F_AssembleByteStream(
	pSrc:= ADR(SIR.Code), 
	SrcLen:= INT_TO_UDINT(LEN(SIR.Code)), 
	pDest:= ADR(SendTelegram), 
	DestLen:= SIZEOF(SendTelegram), 
	WritePointer:= WritePointer);

F_AssembleByteStream(
	pSrc:= ADR(SIR.TU_ID), 
	SrcLen:= INT_TO_UDINT(LEN(SIR.TU_ID)), 
	pDest:= ADR(SendTelegram), 
	DestLen:= SIZEOF(SendTelegram), 
	WritePointer:= WritePointer);	
	
F_AssembleByteStream(
	pSrc:= ADR(SIR.Counter1), 
	SrcLen:= INT_TO_UDINT(LEN(SIR.Counter1)), 
	pDest:= ADR(SendTelegram), 
	DestLen:= SIZEOF(SendTelegram), 
	WritePointer:= WritePointer);	
	
F_AssembleByteStream(
	pSrc:= ADR(SIR.Counter2), 
	SrcLen:= INT_TO_UDINT(LEN(SIR.Counter2)), 
	pDest:= ADR(SendTelegram), 
	DestLen:= SIZEOF(SendTelegram), 
	WritePointer:= WritePointer);	
	
F_AssembleByteStream(
	pSrc:= ADR(SIR.Counter3), 
	SrcLen:= INT_TO_UDINT(LEN(SIR.Counter3)), 
	pDest:= ADR(SendTelegram), 
	DestLen:= SIZEOF(SendTelegram), 
	WritePointer:= WritePointer);	
	
F_AssembleByteStream(
	pSrc:= ADR(SIR.Counter4), 
	SrcLen:= INT_TO_UDINT(LEN(SIR.Counter4)), 
	pDest:= ADR(SendTelegram), 
	DestLen:= SIZEOF(SendTelegram), 
	WritePointer:= WritePointer);	
	
F_AssembleByteStream(
	pSrc:= ADR(SIR.Counter5), 
	SrcLen:= INT_TO_UDINT(LEN(SIR.Counter5)), 
	pDest:= ADR(SendTelegram), 
	DestLen:= SIZEOF(SendTelegram), 
	WritePointer:= WritePointer);	

F_AssembleByteStream(
	pSrc:= ADR(SIR.ReturnCode), 
	SrcLen:= INT_TO_UDINT(LEN(SIR.ReturnCode)), 
	pDest:= ADR(SendTelegram), 
	DestLen:= SIZEOF(SendTelegram), 
	WritePointer:= WritePointer);


// Add to buffer of Base Driver
M_ProcessSIR := fbBaseDriver.M_SendAppData(
					mpSendData := ADR(SendTelegram),
					mSendDataLen := WritePointer);

// Forward to mirror channel
M_MirrorData(Data := ADR(SendTelegram), DataLen := WritePointer);
END_METHOD

METHOD PROTECTED M_ProcessSNR : BOOL
(**************************************************************************************
 * 	Application		:	BoxControl Framework
 *	Revision		:	$Revision: 404529 $
 *	Revision date	:	$Date: 2018-04-23 08:21:38 +0200 (Mo., 23 Apr 2018) $
 *	Last changed by	:	$Author: b7bolm $
 *	URL				:	$URL: http://almscdc.swisslog.com/repo/SWPD/Development/BoxControlFramework/20_Release/trunk/01_Software/BCF/BCF/JumpStart/20_Product/10_App/11_Com/10_Lib/10_Conv/12_MFCS/11_SIS/FB_SIS_MsgManager_6_1.TcPOU $
 *
 *	Purpose			:	Send SNR
 *
 * ------------------------------------------------------------------------------------
 *	Copyright Swisslog [IP AG], Switzerland. All rights reserved.
 * 
 * ------------------------------------------------------------------------------------
 *	
 * 	Revision History: 
 *
 * 	VERSION			DATE			INITIALS			DESCRIPTION
 *	0.1				01.01.2001		swl					Example
 *
 **************************************************************************************)
VAR_INPUT
 	meChannelSrc		: E_MFCS_Channel; // Source communicaton channel
	mpSNR				: POINTER TO ST_ITC_SNR; // Pointer to SNR
END_VAR
(**************************************************************************************************************
 	Check if a telegram needs to be send
***************************************************************************************************************)
// If settings allow sending a SNR 	
IF  Settings.Telegrams.SendSNR THEN
	// If the source of the request is this channel or is undefined
	IF meChannelSrc = Settings.MFCS_Channel OR
		meChannelSrc = E_MFCS_Channel.BEGIN_CHANNEL THEN
		;//Proceed
	ELSE // Source is a different MFCS Connection
		// Dont send a telegram		
		RETURN;
	END_IF	
ELSE
	// Dont send a telegram		
	RETURN;
END_IF

(**************************************************************************************************************
 	ITC - Map generic data to type
***************************************************************************************************************)
MEMCPY(destAddr := ADR(SNR_ITC), srcAddr := mpSNR, n := SIZEOF(SNR_ITC));

(**************************************************************************************************************
 	Formatting data
***************************************************************************************************************)

// Get SIS-Number 
SNR.Position := F_StuffString(
					InputString 	:= SNR_ITC.Position, 
					StringLength	:= SIS_6_1.POSITION_STRINGLENGTH, 
					StuffCharacter 	:= '0',
					LeftAligned		:= FALSE);

// Get TU-ID 
SNR.TU_ID := F_StuffString(
				InputString 	:= SNR_ITC.TU_ID, 
				StringLength	:= SIS_6_1.TU_ID_STRINGLENGTH, 
				StuffCharacter 	:= ' ',
				LeftAligned		:= FALSE);


// Get Error Code 
SNR.InfoCode := F_StuffString(
					InputString 	:= INT_TO_STRING(SNR_ITC.InfoCode), 
					StringLength	:= SIS_6_1.ERRORCODE_STRINGLENGTH, 
					StuffCharacter 	:= '0',
					LeftAligned		:= FALSE);
					
					
(**************************************************************************************************************
 	Build string and add to Base Driver
***************************************************************************************************************)
MEMSET(destAddr := ADR(SendTelegram), 0, SIZEOF(SendTelegram));
WritePointer := 0;

F_AssembleByteStream(
	pSrc:= ADR('SNR'), 
	SrcLen:= 3, 
	pDest:= ADR(SendTelegram), 
	DestLen:= SIZEOF(SendTelegram), 
	WritePointer:= WritePointer);
	
F_AssembleByteStream(
	pSrc:= ADR(SNR.Position), 
	SrcLen:= INT_TO_UDINT(LEN(SNR.Position)), 
	pDest:= ADR(SendTelegram), 
	DestLen:= SIZEOF(SendTelegram), 
	WritePointer:= WritePointer);

F_AssembleByteStream(
	pSrc:= ADR(SNR.TU_ID), 
	SrcLen:= INT_TO_UDINT(LEN(SNR.TU_ID)), 
	pDest:= ADR(SendTelegram), 
	DestLen:= SIZEOF(SendTelegram), 
	WritePointer:= WritePointer);
	
F_AssembleByteStream(
	pSrc:= ADR(SNR.InfoCode), 
	SrcLen:= INT_TO_UDINT(LEN(SNR.InfoCode)), 
	pDest:= ADR(SendTelegram), 
	DestLen:= SIZEOF(SendTelegram), 
	WritePointer:= WritePointer);

// Add to buffer of Base Driver
M_ProcessSNR := fbBaseDriver.M_SendAppData(
					mpSendData := ADR(SendTelegram),
					mSendDataLen := WritePointer);

// Forward to mirror channel
M_MirrorData(Data := ADR(SendTelegram), DataLen := WritePointer);
END_METHOD

METHOD PROTECTED M_ProcessSSR : BOOL
(**************************************************************************************
 * 	Application		:	BoxControl Framework
 *	Revision		:	$Revision: 404529 $
 *	Revision date	:	$Date: 2018-04-23 08:21:38 +0200 (Mo., 23 Apr 2018) $
 *	Last changed by	:	$Author: b7bolm $
 *	URL				:	$URL: http://almscdc.swisslog.com/repo/SWPD/Development/BoxControlFramework/20_Release/trunk/01_Software/BCF/BCF/JumpStart/20_Product/10_App/11_Com/10_Lib/10_Conv/12_MFCS/11_SIS/FB_SIS_MsgManager_6_1.TcPOU $
 *
 *	Purpose			:	Send SSR
 *
 * ------------------------------------------------------------------------------------
 *	Copyright Swisslog [IP AG], Switzerland. All rights reserved.
 * 
 * ------------------------------------------------------------------------------------
 *	
 * 	Revision History: 
 *
 * 	VERSION			DATE			INITIALS			DESCRIPTION
 *	0.1				01.01.2001		swl					Example
 *
 **************************************************************************************)
VAR_INPUT
 	meChannelSrc		: E_MFCS_Channel; // Source communicaton channel
	mpSSR				: POINTER TO ST_ITC_SSR; // Pointer to SSR
END_VAR
(**************************************************************************************************************
 	Check if a telegram needs to be send
***************************************************************************************************************)
// If settings allow sending a SSR 	
IF  Settings.Telegrams.SendSSR THEN
	// If the source of the request is this channel or is undefined
	IF meChannelSrc = Settings.MFCS_Channel OR
		meChannelSrc = E_MFCS_Channel.BEGIN_CHANNEL THEN
		;//Proceed
	ELSE // Source is a different MFCS Connection
		// Dont send a telegram		
		RETURN;
	END_IF	
ELSE
	// Dont send a telegram		
	RETURN;
END_IF

(**************************************************************************************************************
 	ITC - Map generic data to type
***************************************************************************************************************)
MEMCPY(destAddr := ADR(SSR_ITC), srcAddr := mpSSR, n := SIZEOF(SSR_ITC));

(**************************************************************************************************************
 	Formatting data
***************************************************************************************************************)
// Get Subsystem name 
SSR.SubsystemName := F_StuffString(
						InputString 	:= SSR_ITC.SubsystemName, 
						StringLength	:= SIS_6_1.POSITION_STRINGLENGTH, 
						StuffCharacter 	:= '0',
						LeftAligned		:= FALSE);

// Get Mode 
SSR.Mode := INT_TO_STRING(SSR_ITC.eMode);

// Get system info
SSR.State := INT_TO_STRING(SSR_ITC.eState);

// Get system info
SSR.SystemInfo := INT_TO_STRING(SSR_ITC.eSystemInfo);

// Get ErrorState 
SSR.ErrorState := INT_TO_STRING(SSR_ITC.eErrorState);

// Get ErrorCode 
SSR.ErrorCode := F_StuffString(
					InputString 	:= INT_TO_STRING(SSR_ITC.eErrorCode), 
					StringLength	:= SIS_6_1.ERRORCODE_STRINGLENGTH, 
					StuffCharacter 	:= '0',
					LeftAligned		:= FALSE);

// Get ErrorType 
SSR.ErrorType := INT_TO_STRING(SSR_ITC.eErrorType);

// Get ErrorInformation 
SSR.ErrorInformation := F_StuffString(
							InputString 	:= SSR_ITC.ErrorInformation, 
							StringLength	:= SIS_6_1.ERRORINFORMATION_STRINGLENGTH, 
							StuffCharacter 	:= ' ',
							LeftAligned		:= TRUE);

// Get Variable 
SSR.Variable := F_StuffString(
					InputString 	:= DINT_TO_STRING(SSR_ITC.Variable), 
					StringLength	:= SIS_6_1.CONTROLVARIABLE_STRINGLENGTH, 
					StuffCharacter 	:= '0',
					LeftAligned		:= FALSE);

// Get Error Code 
SSR.ReturnCode := F_StuffString(
					InputString 	:= INT_TO_STRING(SSR_ITC.eReturnCode), 
					StringLength	:= SIS_6_1.ERRORCODE_STRINGLENGTH, 
					StuffCharacter 	:= '0',
					LeftAligned		:= FALSE);


(**************************************************************************************************************
 	Build string and add to Base Driver
***************************************************************************************************************)
MEMSET(destAddr := ADR(SendTelegram), 0, SIZEOF(SendTelegram));
WritePointer := 0;

F_AssembleByteStream(
	pSrc:= ADR('SSR'), 
	SrcLen:= 3, 
	pDest:= ADR(SendTelegram), 
	DestLen:= SIZEOF(SendTelegram), 
	WritePointer:= WritePointer);
	
F_AssembleByteStream(
	pSrc:= ADR(SSR.SubsystemName), 
	SrcLen:= INT_TO_UDINT(LEN(SSR.SubsystemName)), 
	pDest:= ADR(SendTelegram), 
	DestLen:= SIZEOF(SendTelegram), 
	WritePointer:= WritePointer);

F_AssembleByteStream(
	pSrc:= ADR(SSR.Mode), 
	SrcLen:= INT_TO_UDINT(LEN(SSR.Mode)), 
	pDest:= ADR(SendTelegram), 
	DestLen:= SIZEOF(SendTelegram), 
	WritePointer:= WritePointer);	

F_AssembleByteStream(
	pSrc:= ADR(SSR.State), 
	SrcLen:= INT_TO_UDINT(LEN(SSR.State)), 
	pDest:= ADR(SendTelegram), 
	DestLen:= SIZEOF(SendTelegram), 
	WritePointer:= WritePointer);	

F_AssembleByteStream(
	pSrc:= ADR(SSR.SystemInfo), 
	SrcLen:= INT_TO_UDINT(LEN(SSR.SystemInfo)), 
	pDest:= ADR(SendTelegram), 
	DestLen:= SIZEOF(SendTelegram), 
	WritePointer:= WritePointer);	
	
F_AssembleByteStream(
	pSrc:= ADR(SSR.ErrorState), 
	SrcLen:= INT_TO_UDINT(LEN(SSR.ErrorState)), 
	pDest:= ADR(SendTelegram), 
	DestLen:= SIZEOF(SendTelegram), 
	WritePointer:= WritePointer);

F_AssembleByteStream(
	pSrc:= ADR(SSR.ErrorCode), 
	SrcLen:= INT_TO_UDINT(LEN(SSR.ErrorCode)), 
	pDest:= ADR(SendTelegram), 
	DestLen:= SIZEOF(SendTelegram), 
	WritePointer:= WritePointer);

F_AssembleByteStream(
	pSrc:= ADR(SSR.ErrorType), 
	SrcLen:= INT_TO_UDINT(LEN(SSR.ErrorType)), 
	pDest:= ADR(SendTelegram), 
	DestLen:= SIZEOF(SendTelegram), 
	WritePointer:= WritePointer);
	
F_AssembleByteStream(
	pSrc:= ADR(SSR.ErrorInformation), 
	SrcLen:= INT_TO_UDINT(LEN(SSR.ErrorInformation)), 
	pDest:= ADR(SendTelegram), 
	DestLen:= SIZEOF(SendTelegram), 
	WritePointer:= WritePointer);
	
F_AssembleByteStream(
	pSrc:= ADR(SSR.Variable), 
	SrcLen:= INT_TO_UDINT(LEN(SSR.Variable)), 
	pDest:= ADR(SendTelegram), 
	DestLen:= SIZEOF(SendTelegram), 
	WritePointer:= WritePointer);
	
F_AssembleByteStream(
	pSrc:= ADR(SSR.ReturnCode), 
	SrcLen:= INT_TO_UDINT(LEN(SSR.ReturnCode)), 
	pDest:= ADR(SendTelegram), 
	DestLen:= SIZEOF(SendTelegram), 
	WritePointer:= WritePointer);

// Add to buffer of Base Driver
M_ProcessSSR := fbBaseDriver.M_SendAppData(
					mpSendData := ADR(SendTelegram),
					mSendDataLen := WritePointer);

// Forward to mirror channel
M_MirrorData(Data := ADR(SendTelegram), DataLen := WritePointer);
END_METHOD

METHOD PROTECTED M_ProcessTDR : BOOL
(**************************************************************************************
 * 	Application		:	BoxControl Framework
 *	Revision		:	$Revision: 404529 $
 *	Revision date	:	$Date: 2018-04-23 08:21:38 +0200 (Mo., 23 Apr 2018) $
 *	Last changed by	:	$Author: b7bolm $
 *	URL				:	$URL: http://almscdc.swisslog.com/repo/SWPD/Development/BoxControlFramework/20_Release/trunk/01_Software/BCF/BCF/JumpStart/20_Product/10_App/11_Com/10_Lib/10_Conv/12_MFCS/11_SIS/FB_SIS_MsgManager_6_1.TcPOU $
 *
 *	Purpose			:	Send TDR
 *
 * ------------------------------------------------------------------------------------
 *	Copyright Swisslog [IP AG], Switzerland. All rights reserved.
 * 
 * ------------------------------------------------------------------------------------
 *	
 * 	Revision History: 
 *
 * 	VERSION			DATE			INITIALS			DESCRIPTION
 *	0.1				01.01.2001		swl					Example
 *
 **************************************************************************************)
VAR_INPUT
 	meChannelSrc		: E_MFCS_Channel; // Source communicaton channel
	mpTDR				: POINTER TO ST_ITC_TDR; // Pointer to TDR
END_VAR
(**************************************************************************************************************
 	Check if a telegram needs to be send
***************************************************************************************************************)
// If settings allow sending a TDR 	
IF  Settings.Telegrams.SendTDR THEN
	// If the source of the request is this channel or is undefined
	IF meChannelSrc = Settings.MFCS_Channel OR
		meChannelSrc = E_MFCS_Channel.BEGIN_CHANNEL THEN
		;//Proceed
	ELSE // Source is a different MFCS Connection
		// Dont send a telegram		
		RETURN;
	END_IF	
ELSE
	// Dont send a telegram		
	RETURN;
END_IF

(**************************************************************************************************************
 	ITC - Map generic data to type
***************************************************************************************************************)
MEMCPY(destAddr := ADR(TDR_ITC), srcAddr := mpTDR, n := SIZEOF(TDR_ITC));

(**************************************************************************************************************
 	Formatting data
***************************************************************************************************************)
// Get SIS-Number 
TDR.Position := F_StuffString(
					InputString 	:= TDR_ITC.Position, 
					StringLength	:= SIS_6_1.POSITION_STRINGLENGTH, 
					StuffCharacter 	:= '0',
					LeftAligned		:= FALSE);

// Get TU-ID 
TDR.TU_ID := F_StuffString(
				InputString 	:= TDR_ITC.TU_ID, 
				StringLength	:= SIS_6_1.TU_ID_STRINGLENGTH, 
				StuffCharacter 	:= ' ',
				LeftAligned		:= FALSE);
					
// Get Assignment 
TDR.AssignmentID := F_StuffString(
						InputString 	:= UDINT_TO_STRING(TDR_ITC.AssignmentID), 
						StringLength	:= SIS_6_1.ASSIGNMENT_ID_STRINGLENGTH, 
						StuffCharacter 	:= '0',
						LeftAligned		:= FALSE);

// Get MSG Sequence 
TDR.MsgSequence := 	F_StuffString(
						InputString 	:= INT_TO_STRING(TDR_ITC.MsgSequence), 
						StringLength	:= SIS_6_1.MSG_SEQUENCE_STRINGLENGTH, 
						StuffCharacter 	:= '0',
						LeftAligned		:= FALSE);

// Get return Code 
TDR.ReturnCode := F_StuffString(
					InputString 	:= INT_TO_STRING(TDR_ITC.ReturnCode), 
					StringLength	:= SIS_6_1.ERRORCODE_STRINGLENGTH, 
					StuffCharacter 	:= '0',
					LeftAligned		:= FALSE);



(**************************************************************************************************************
 	Build string and add to Base Driver
***************************************************************************************************************)
MEMSET(destAddr := ADR(SendTelegram), 0, SIZEOF(SendTelegram));
WritePointer := 0;

F_AssembleByteStream(
	pSrc:= ADR('TDR'), 
	SrcLen:= 3, 
	pDest:= ADR(SendTelegram), 
	DestLen:= SIZEOF(SendTelegram), 
	WritePointer:= WritePointer);
	
F_AssembleByteStream(
	pSrc:= ADR(TDR.Position), 
	SrcLen:= INT_TO_UDINT(LEN(TDR.Position)), 
	pDest:= ADR(SendTelegram), 
	DestLen:= SIZEOF(SendTelegram), 
	WritePointer:= WritePointer);

F_AssembleByteStream(
	pSrc:= ADR(TDR.TU_ID), 
	SrcLen:= INT_TO_UDINT(LEN(TDR.TU_ID)), 
	pDest:= ADR(SendTelegram), 
	DestLen:= SIZEOF(SendTelegram), 
	WritePointer:= WritePointer);
	
F_AssembleByteStream(
	pSrc:= ADR(TDR.AssignmentID), 
	SrcLen:= INT_TO_UDINT(LEN(TDR.AssignmentID)), 
	pDest:= ADR(SendTelegram), 
	DestLen:= SIZEOF(SendTelegram), 
	WritePointer:= WritePointer);
	
F_AssembleByteStream(
	pSrc:= ADR(TDR.MsgSequence), 
	SrcLen:= INT_TO_UDINT(LEN(TDR.MsgSequence)), 
	pDest:= ADR(SendTelegram), 
	DestLen:= SIZEOF(SendTelegram), 
	WritePointer:= WritePointer);	
	
F_AssembleByteStream(
	pSrc:= ADR(TDR.ReturnCode), 
	SrcLen:= INT_TO_UDINT(LEN(TDR.ReturnCode)), 
	pDest:= ADR(SendTelegram), 
	DestLen:= SIZEOF(SendTelegram), 
	WritePointer:= WritePointer);	

// Add to buffer of Base Driver
M_ProcessTDR := fbBaseDriver.M_SendAppData(
					mpSendData := ADR(SendTelegram),
					mSendDataLen := WritePointer);

// Forward to mirror channel
M_MirrorData(Data := ADR(SendTelegram), DataLen := WritePointer);
END_METHOD

METHOD PROTECTED M_ProcessTTC : BOOL
(**************************************************************************************
 * 	Application		:	BoxControl Framework
 *	Revision		:	$Revision: 404529 $
 *	Revision date	:	$Date: 2018-04-23 08:21:38 +0200 (Mo., 23 Apr 2018) $
 *	Last changed by	:	$Author: b7bolm $
 *	URL				:	$URL: http://almscdc.swisslog.com/repo/SWPD/Development/BoxControlFramework/20_Release/trunk/01_Software/BCF/BCF/JumpStart/20_Product/10_App/11_Com/10_Lib/10_Conv/12_MFCS/11_SIS/FB_SIS_MsgManager_6_1.TcPOU $
 *
 *	Purpose			:	Send TTC
 *
 * ------------------------------------------------------------------------------------
 *	Copyright Swisslog [IP AG], Switzerland. All rights reserved.
 * 
 * ------------------------------------------------------------------------------------
 *	
 * 	Revision History: 
 *
 * 	VERSION			DATE			INITIALS			DESCRIPTION
 *	0.1				01.01.2001		swl					Example
 *
 **************************************************************************************)
VAR_INPUT
 	meChannelSrc		: E_MFCS_Channel; // Source communicaton channel
	mpTTC				: POINTER TO ST_ITC_TTC; // Pointer to TTC
END_VAR
(**************************************************************************************************************
 	Check if a telegram needs to be send
***************************************************************************************************************)
// If settings allow sending a TTC 	
IF  Settings.Telegrams.SendTTC THEN
	// If the source of the request is this channel or is undefined
	IF meChannelSrc = Settings.MFCS_Channel OR
		meChannelSrc = E_MFCS_Channel.BEGIN_CHANNEL THEN
		;//Proceed
	ELSE // Source is a different MFCS Connection
		// Dont send a telegram		
		RETURN;
	END_IF	
ELSE
	// Dont send a telegram		
	RETURN;
END_IF

(**************************************************************************************************************
 	ITC - Map generic data to type
***************************************************************************************************************)
MEMCPY(destAddr := ADR(TTC_ITC), srcAddr := mpTTC, n := SIZEOF(TTC_ITC));

(**************************************************************************************************************
 	Formatting data
***************************************************************************************************************)
// Get SIS-Number 
TTC.Position := F_StuffString(
					InputString 	:= TTC_ITC.Position, 
					StringLength	:= SIS_6_1.POSITION_STRINGLENGTH, 
					StuffCharacter 	:= '0',
					LeftAligned		:= FALSE);

// Get TU-DataIndex 
TTC.TU_DataIndex := F_StuffString(
						InputString 	:= DINT_TO_STRING(TTC_ITC.TU_DataIndex), 
						StringLength	:= SIS_6_1.TU_DATAINDEX_STRINGLENGTH, 
						StuffCharacter 	:= '0',
						LeftAligned		:= FALSE);

// Get MSG Sequence 
TTC.MsgSequence := F_StuffString(
						InputString 	:= INT_TO_STRING(TTC_ITC.MsgSequence), 
						StringLength	:= SIS_6_1.MSG_SEQUENCE_STRINGLENGTH, 
						StuffCharacter 	:= '0',
						LeftAligned		:= FALSE);

// Get TU-ID 
TTC.TU_ID := F_StuffString(
				InputString 	:= TTC_ITC.TU_ID, 
				StringLength	:= SIS_6_1.TU_ID_STRINGLENGTH, 
				StuffCharacter 	:= ' ',
				LeftAligned		:= FALSE);
				
// Get Assignment 
TTC.AssignmentID := F_StuffString(
						InputString 	:= UDINT_TO_STRING(TTC_ITC.AssignmentID), 
						StringLength	:= SIS_6_1.ASSIGNMENT_ID_STRINGLENGTH, 
						StuffCharacter 	:= '0',
						LeftAligned		:= FALSE);

// Get Error Code 
TTC.ReturnCode := F_StuffString(
					InputString 	:= INT_TO_STRING(TTC_ITC.ReturnCode), 
					StringLength	:= SIS_6_1.ERRORCODE_STRINGLENGTH, 
					StuffCharacter 	:= '0',
					LeftAligned		:= FALSE);

(**************************************************************************************************************
 	Build string and add to Base Driver
***************************************************************************************************************)
MEMSET(destAddr := ADR(SendTelegram), 0, SIZEOF(SendTelegram));
WritePointer := 0;

F_AssembleByteStream(
	pSrc:= ADR('TTC'), 
	SrcLen:= 3, 
	pDest:= ADR(SendTelegram), 
	DestLen:= SIZEOF(SendTelegram), 
	WritePointer:= WritePointer);
	
F_AssembleByteStream(
	pSrc:= ADR(TTC.Position), 
	SrcLen:= INT_TO_UDINT(LEN(TTC.Position)), 
	pDest:= ADR(SendTelegram), 
	DestLen:= SIZEOF(SendTelegram), 
	WritePointer:= WritePointer);
	
F_AssembleByteStream(
	pSrc:= ADR(TTC.TU_DataIndex), 
	SrcLen:= INT_TO_UDINT(LEN(TTC.TU_DataIndex)), 
	pDest:= ADR(SendTelegram), 
	DestLen:= SIZEOF(SendTelegram), 
	WritePointer:= WritePointer);
	
F_AssembleByteStream(
	pSrc:= ADR(TTC.MsgSequence), 
	SrcLen:= INT_TO_UDINT(LEN(TTC.MsgSequence)), 
	pDest:= ADR(SendTelegram), 
	DestLen:= SIZEOF(SendTelegram), 
	WritePointer:= WritePointer);

F_AssembleByteStream(
	pSrc:= ADR(TTC.TU_ID), 
	SrcLen:= INT_TO_UDINT(LEN(TTC.TU_ID)), 
	pDest:= ADR(SendTelegram), 
	DestLen:= SIZEOF(SendTelegram), 
	WritePointer:= WritePointer);

F_AssembleByteStream(
	pSrc:= ADR(TTC.AssignmentID), 
	SrcLen:= INT_TO_UDINT(LEN(TTC.AssignmentID)), 
	pDest:= ADR(SendTelegram), 
	DestLen:= SIZEOF(SendTelegram), 
	WritePointer:= WritePointer);

F_AssembleByteStream(
	pSrc:= ADR(TTC.ReturnCode), 
	SrcLen:= INT_TO_UDINT(LEN(TTC.ReturnCode)), 
	pDest:= ADR(SendTelegram), 
	DestLen:= SIZEOF(SendTelegram), 
	WritePointer:= WritePointer);

// Add to buffer of Base Driver
M_ProcessTTC := fbBaseDriver.M_SendAppData(
					mpSendData := ADR(SendTelegram),
					mSendDataLen := WritePointer);

// Forward to mirror channel
M_MirrorData(Data := ADR(SendTelegram), DataLen := WritePointer);
END_METHOD

METHOD PROTECTED M_ProcessTTQ : BOOL
(**************************************************************************************
 * 	Application		:	BoxControl Framework
 *	Revision		:	$Revision: 404529 $
 *	Revision date	:	$Date: 2018-04-23 08:21:38 +0200 (Mo., 23 Apr 2018) $
 *	Last changed by	:	$Author: b7bolm $
 *	URL				:	$URL: http://almscdc.swisslog.com/repo/SWPD/Development/BoxControlFramework/20_Release/trunk/01_Software/BCF/BCF/JumpStart/20_Product/10_App/11_Com/10_Lib/10_Conv/12_MFCS/11_SIS/FB_SIS_MsgManager_6_1.TcPOU $
 *
 *	Purpose			:	Send TTQ
 *
 * ------------------------------------------------------------------------------------
 *	Copyright Swisslog [IP AG], Switzerland. All rights reserved.
 * 
 * ------------------------------------------------------------------------------------
 *	
 * 	Revision History: 
 *
 * 	VERSION			DATE			INITIALS			DESCRIPTION
 *	0.1				01.01.2001		swl					Example
 *
 **************************************************************************************)
VAR_INPUT
 	meChannelSrc		: E_MFCS_Channel; // Source communicaton channel
	mpTTQ				: POINTER TO ST_ITC_TTQ; // Pointer to TTQ
END_VAR
(**************************************************************************************************************
 	Check if a telegram needs to be send
***************************************************************************************************************)
// If settings allow sending a TTQ 	
IF  Settings.Telegrams.SendTTQ THEN
	// If the source of the request is this channel or is undefined
	IF meChannelSrc = Settings.MFCS_Channel OR
		meChannelSrc = E_MFCS_Channel.BEGIN_CHANNEL THEN
		;//Proceed
	ELSE // Source is a different MFCS Connection
		// Dont send a telegram		
		RETURN;
	END_IF	
ELSE
	// Dont send a telegram		
	RETURN;
END_IF

(**************************************************************************************************************
 	ITC - Map generic data to type
***************************************************************************************************************)
MEMCPY(destAddr := ADR(TTQ_ITC), srcAddr := mpTTQ, n := SIZEOF(TTQ_ITC));

(**************************************************************************************************************
 	Formatting data
***************************************************************************************************************)
// Get SIS-Number 
TTQ.Position := F_StuffString(
					InputString 	:= TTQ_ITC.Position, 
					StringLength	:= SIS_6_1.POSITION_STRINGLENGTH, 
					StuffCharacter 	:= '0',
					LeftAligned		:= FALSE);

// Get TU-DataIndex 
TTQ.TU_DataIndex := F_StuffString(
						InputString 	:= DINT_TO_STRING(TTQ_ITC.TU_DataIndex), 
						StringLength	:= SIS_6_1.TU_DATAINDEX_STRINGLENGTH, 
						StuffCharacter 	:= '0',
						LeftAligned		:= FALSE);

// Get TU-ID 
TTQ.TU_ID := F_StuffString(
				InputString 	:= TTQ_ITC.TU_ID, 
				StringLength	:= SIS_6_1.TU_ID_STRINGLENGTH, 
				StuffCharacter 	:= ' ',
				LeftAligned		:= FALSE);

// Get Number of TT's 
TTQ.NbrOfTT :=  F_StuffString(
						InputString 	:= INT_TO_STRING(TTQ_ITC.NbrOfTT), 
						StringLength	:= SIS_6_1.TTQ_NUMBER_OF_TT_STRINGLENGTH, 
						StuffCharacter 	:= '0',
						LeftAligned		:= FALSE);

// Get Label Length						
TTQ.Label := F_StuffString(
				InputString 	:= TTQ_ITC.Label, 
				StringLength	:= Conveyor.LABEL_LENGTH, 
				StuffCharacter 	:= '-',
				LeftAligned		:= FALSE);

(**************************************************************************************************************
 	Build string and add to Base Driver
***************************************************************************************************************)
MEMSET(destAddr := ADR(SendTelegram), 0, SIZEOF(SendTelegram));
WritePointer := 0;

F_AssembleByteStream(
	pSrc:= ADR('TTQ'), 
	SrcLen:= 3, 
	pDest:= ADR(SendTelegram), 
	DestLen:= SIZEOF(SendTelegram), 
	WritePointer:= WritePointer);
	
F_AssembleByteStream(
	pSrc:= ADR(TTQ .Position), 
	SrcLen:= INT_TO_UDINT(LEN(TTQ.Position)), 
	pDest:= ADR(SendTelegram), 
	DestLen:= SIZEOF(SendTelegram), 
	WritePointer:= WritePointer);

F_AssembleByteStream(
	pSrc:= ADR(TTQ.TU_DataIndex), 
	SrcLen:= INT_TO_UDINT(LEN(TTQ.TU_DataIndex)), 
	pDest:= ADR(SendTelegram), 
	DestLen:= SIZEOF(SendTelegram), 
	WritePointer:= WritePointer);
	
F_AssembleByteStream(
	pSrc:= ADR(TTQ.TU_ID), 
	SrcLen:= INT_TO_UDINT(LEN(TTQ.TU_ID)), 
	pDest:= ADR(SendTelegram), 
	DestLen:= SIZEOF(SendTelegram), 
	WritePointer:= WritePointer);
	
F_AssembleByteStream(
	pSrc:= ADR(TTQ.NbrOfTT), 
	SrcLen:= INT_TO_UDINT(LEN(TTQ.NbrOfTT)), 
	pDest:= ADR(SendTelegram), 
	DestLen:= SIZEOF(SendTelegram), 
	WritePointer:= WritePointer);
	
F_AssembleByteStream(
	pSrc:= ADR(TTQ.Label), 
	SrcLen:= INT_TO_UDINT(LEN(TTQ.Label)), 
	pDest:= ADR(SendTelegram), 
	DestLen:= SIZEOF(SendTelegram), 
	WritePointer:= WritePointer);	


// Add to buffer of Base Driver
M_ProcessTTQ := fbBaseDriver.M_SendAppData(
					mpSendData := ADR(SendTelegram),
					mSendDataLen := WritePointer);

// Forward to mirror channel
M_MirrorData(Data := ADR(SendTelegram), DataLen := WritePointer);
END_METHOD

METHOD PROTECTED M_ProcessTUR : BOOL
(**************************************************************************************
 * 	Application		:	BoxControl Framework
 *	Revision		:	$Revision: 415970 $
 *	Revision date	:	$Date: 2018-10-24 16:08:06 +0200 (Mi., 24 Okt 2018) $
 *	Last changed by	:	$Author: d7herza $
 *	URL				:	$URL: http://almscdc.swisslog.com/repo/SWPD/Development/BoxControlFramework/20_Release/branches/R1.5.x/01_Software/BCF/BCF/JumpStart/20_Product/10_App/11_Com/10_Lib/10_Conv/12_MFCS/11_SIS/FB_SIS_MsgManager_6_1.TcPOU $
 *
 *	Purpose			:	Send TUR
 *
 * ------------------------------------------------------------------------------------
 *	Copyright Swisslog [IP AG], Switzerland. All rights reserved.
 * 
 * ------------------------------------------------------------------------------------
 *	
 * 	Revision History: 
 *
 * 	VERSION			DATE			INITIALS			DESCRIPTION
 *	0.1				01.01.2001		swl					Example
 *
 *************************************************************************************)
VAR_INPUT
 	meChannelSrc		: E_MFCS_Channel; // Source communicaton channel
	mpTUR				: POINTER TO ST_ITC_TUR; // Pointer to TUR
END_VAR

VAR
	DestinationIdx			: INT; // Iterator
END_VAR
(**************************************************************************************************************
 	Check if a telegram needs to be send
***************************************************************************************************************)
// If settings allow sending a TUR 	
IF  Settings.Telegrams.SendTUR THEN
	// If the source of the request is this channel or is undefined
	IF meChannelSrc = Settings.MFCS_Channel OR
		meChannelSrc = E_MFCS_Channel.BEGIN_CHANNEL THEN
		;//Proceed
	ELSE // Source is a different MFCS Connection
		// Dont send a telegram		
		RETURN;
	END_IF	
ELSE
	// Dont send a telegram		
	RETURN;
END_IF

(**************************************************************************************************************
 	ITC - Map generic data to type
***************************************************************************************************************)
MEMCPY(destAddr := ADR(TUR_ITC), srcAddr := mpTUR, n := SIZEOF(TUR_ITC));

(**************************************************************************************************************
 	Formatting data
***************************************************************************************************************)
// Get SIS-Number 
TUR.Position := F_StuffString(
					InputString 	:= TUR_ITC.Position, 
					StringLength	:= SIS_6_1.POSITION_STRINGLENGTH, 
					StuffCharacter 	:= '0',
					LeftAligned		:= FALSE);
				
// Get TU-Data index
TUR.TU_DataIndex := F_StuffString(
				InputString 	:= DINT_TO_STRING(TUR_ITC.TU_DataIndex), 
				StringLength	:= SIS_6_1.TU_DATAINDEX_STRINGLENGTH, 
				StuffCharacter 	:= '0',
				LeftAligned		:= FALSE);
				
// Get TU-ID 
TUR.TU_ID := F_StuffString(
				InputString 	:= TUR_ITC.TU_ID, 
				StringLength	:= SIS_6_1.TU_ID_STRINGLENGTH, 
				StuffCharacter 	:= ' ',
				LeftAligned		:= FALSE);

// Get TU-Type 
TUR.TU_Type := 	F_StuffString(
					InputString 	:= INT_TO_STRING(TUR_ITC.TU_Type), 
					StringLength	:= SIS_6_1.TU_TYPE_STRINGLENGTH, 
					StuffCharacter 	:= '0',
					LeftAligned		:= FALSE);
				
// Get Assignment id
TUR.AssignmentID := F_StuffString(
						InputString 	:= UDINT_TO_STRING(TUR_ITC.AssignmentID), 
						StringLength	:= SIS_6_1.ASSIGNMENT_ID_STRINGLENGTH, 
						StuffCharacter 	:= '0',
						LeftAligned		:= FALSE);;

// Get length
TUR.Length := F_StuffString(
				InputString 	:= INT_TO_STRING(TUR_ITC.Length), 
				StringLength	:= SIS_6_1.DIMENSIONS, 
				StuffCharacter 	:= '0',
				LeftAligned		:= FALSE);

// Get width
TUR.Width := F_StuffString(
				InputString 	:= INT_TO_STRING(TUR_ITC.Width), 
				StringLength	:= SIS_6_1.DIMENSIONS, 
				StuffCharacter 	:= '0',
				LeftAligned		:= FALSE);
					
// Get height
TUR.Height := F_StuffString(
				InputString 	:= INT_TO_STRING(TUR_ITC.Height), 
				StringLength	:= SIS_6_1.DIMENSIONS, 
				StuffCharacter 	:= '0',
				LeftAligned		:= FALSE);

// Get weight
TUR.Weight := F_StuffString(
				InputString 	:= DINT_TO_STRING(TUR_ITC.Weight), 
				StringLength	:= SIS_6_1.TTA_WEIGHT, 
				StuffCharacter 	:= '0',
				LeftAligned		:= FALSE);

// Get weight
TUR.Orientation := F_StuffString(
					InputString 	:= TUR_ITC.Orientation, 
					StringLength	:= SIS_6_1.TTA_ORIENTATION, 
					StuffCharacter 	:= '0',
					LeftAligned		:= FALSE);
				
// get TU parameter
TUR.TU_Parameter := F_StuffString(
						InputString 	:= DINT_TO_STRING(TUR_ITC.TU_Parameter), 
						StringLength	:= SIS_6_1.TTA_TU_PARAMETER, 
						StuffCharacter 	:= '0',
						LeftAligned		:= FALSE);
							
// Get I/O Data 
TUR.IO_Data := F_StuffString(
					InputString 	:= INT_TO_STRING(TUR_ITC.IO_Data), 
					StringLength	:= SIS_6_1.TUR_IO_DATA_STRINGLENGTH, 
					StuffCharacter 	:= '0',
					LeftAligned		:= FALSE);

// Get Lower Limit 
TUR.LowerLimit := F_StuffString(
					InputString 	:= DINT_TO_STRING(TUR_ITC.LowerLimit), 
					StringLength	:= SIS_6_1.TUR_LOWERLIMIT_STRINGLENGTH, 
					StuffCharacter 	:= '0',
					LeftAligned		:= FALSE);

// Get Upper Limit 
TUR.UpperLimit := F_StuffString(
					InputString 	:= DINT_TO_STRING(TUR_ITC.UpperLimit), 
					StringLength	:= SIS_6_1.TUR_UPPERLIMIT_STRINGLENGTH, 
					StuffCharacter 	:= '0',
					LeftAligned		:= FALSE);

// Get sequence					
TUR.Sequence := F_StuffString(
					InputString 	:= ULINT_TO_STRING(TUR_ITC.Sequence), 
					StringLength	:= SIS_6_1.SEQUENCE_STRINGLENGTH, 
					StuffCharacter 	:= '0',
					LeftAligned		:= FALSE);

// Get sub sequence
TUR.SubSequence := F_StuffString(
					InputString 	:= DINT_TO_STRING(TUR_ITC.SubSequence), 
					StringLength	:= SIS_6_1.SUBSEQUENCE_STRINGLENGTH, 
					StuffCharacter 	:= '0',
					LeftAligned		:= FALSE);

// Get sequence size					
TUR.SequenceSize := F_StuffString(
					InputString 	:= DINT_TO_STRING(TUR_ITC.SequenceSize), 
					StringLength	:= SIS_6_1.SEQUENCE_SIZE_STRINGLENGTH, 
					StuffCharacter 	:= '0',
					LeftAligned		:= FALSE);

// Get group ID
TUR.GroupID := F_StuffString(
					InputString 	:= ULINT_TO_STRING(TUR_ITC.GroupID), 
					StringLength	:= SIS_6_1.GROUP_ID_STRINGLENGTH, 
					StuffCharacter 	:= '0',
					LeftAligned		:= FALSE);

// Get Group size
TUR.GroupSize := F_StuffString(
					InputString 	:= DINT_TO_STRING(TUR_ITC.GroupSize), 
					StringLength	:= SIS_6_1.GROUP_SIZE_STRINGLENGTH, 
					StuffCharacter 	:= '0',
					LeftAligned		:= FALSE);

// Get destination slot
TUR.DestinationSlot := F_StuffString(
							InputString 	:= INT_TO_STRING(TUR_ITC.DestinationSlot), 
							StringLength	:= SIS_6_1.DESTINATION_SLOT_STRINGLENGTH, 
							StuffCharacter 	:= '0',
							LeftAligned		:= FALSE);			

// Get Error Code 
TUR.ReturnCode := F_StuffString(
					InputString 	:= INT_TO_STRING(TUR_ITC.ReturnCode), 
					StringLength	:= SIS_6_1.ERRORCODE_STRINGLENGTH, 
					StuffCharacter 	:= '0',
					LeftAligned		:= FALSE);

// Get Number of Destinations 
TUR.NumberOfDestinations := F_StuffString(
								InputString 	:= INT_TO_STRING(TUR_ITC.NumberOfDestinations), 
								StringLength	:= SIS_6_1.TUR_NUMBER_OF_DESTINATIONS_STRINGLENGTH, 
								StuffCharacter 	:= '0',
								LeftAligned		:= FALSE);

// Get Destinations 
FOR DestinationIdx := 1 TO TUR_ITC.NumberOfDestinations DO
	TUR.Destination[DestinationIdx] := F_StuffString(
										InputString 	:= TUR_ITC.Destination[DestinationIdx], 
										StringLength	:= SIS_6_1.POSITION_STRINGLENGTH, 
										StuffCharacter 	:= '0',
										LeftAligned		:= FALSE);

END_FOR


(**************************************************************************************************************
 	Build string and add to Base Driver
***************************************************************************************************************)
MEMSET(destAddr := ADR(SendTelegram), 0, SIZEOF(SendTelegram));
WritePointer := 0;

F_AssembleByteStream(
	pSrc:= ADR('TUR'), 
	SrcLen:= 3, 
	pDest:= ADR(SendTelegram), 
	DestLen:= SIZEOF(SendTelegram), 
	WritePointer:= WritePointer);
	
F_AssembleByteStream(
	pSrc:= ADR(TUR.Position), 
	SrcLen:= INT_TO_UDINT(LEN(TUR.Position)), 
	pDest:= ADR(SendTelegram), 
	DestLen:= SIZEOF(SendTelegram), 
	WritePointer:= WritePointer);

F_AssembleByteStream(
	pSrc:= ADR(TUR.TU_DataIndex), 
	SrcLen:= INT_TO_UDINT(LEN(TUR.TU_DataIndex)), 
	pDest:= ADR(SendTelegram), 
	DestLen:= SIZEOF(SendTelegram), 
	WritePointer:= WritePointer);
	
F_AssembleByteStream(
	pSrc:= ADR(TUR.TU_ID), 
	SrcLen:= INT_TO_UDINT(LEN(TUR.TU_ID)), 
	pDest:= ADR(SendTelegram), 
	DestLen:= SIZEOF(SendTelegram), 
	WritePointer:= WritePointer);

F_AssembleByteStream(
	pSrc:= ADR(TUR.TU_Type), 
	SrcLen:= INT_TO_UDINT(LEN(TUR.TU_Type)), 
	pDest:= ADR(SendTelegram), 
	DestLen:= SIZEOF(SendTelegram), 
	WritePointer:= WritePointer);
	
F_AssembleByteStream(
	pSrc:= ADR(TUR.AssignmentID), 
	SrcLen:= INT_TO_UDINT(LEN(TUR.AssignmentID)), 
	pDest:= ADR(SendTelegram), 
	DestLen:= SIZEOF(SendTelegram), 
	WritePointer:= WritePointer);
	
F_AssembleByteStream(
	pSrc:= ADR(TUR.Length), 
	SrcLen:= INT_TO_UDINT(LEN(TUR.Length)), 
	pDest:= ADR(SendTelegram), 
	DestLen:= SIZEOF(SendTelegram), 
	WritePointer:= WritePointer);
	
F_AssembleByteStream(
	pSrc:= ADR(TUR.Width), 
	SrcLen:= INT_TO_UDINT(LEN(TUR.Width)), 
	pDest:= ADR(SendTelegram), 
	DestLen:= SIZEOF(SendTelegram), 
	WritePointer:= WritePointer);
	
F_AssembleByteStream(
	pSrc:= ADR(TUR.Height), 
	SrcLen:= INT_TO_UDINT(LEN(TUR.Height)), 
	pDest:= ADR(SendTelegram), 
	DestLen:= SIZEOF(SendTelegram), 
	WritePointer:= WritePointer);
	
F_AssembleByteStream(
	pSrc:= ADR(TUR.Weight), 
	SrcLen:= INT_TO_UDINT(LEN(TUR.Weight)), 
	pDest:= ADR(SendTelegram), 
	DestLen:= SIZEOF(SendTelegram), 
	WritePointer:= WritePointer);

F_AssembleByteStream(
	pSrc:= ADR(TUR.Orientation), 
	SrcLen:= INT_TO_UDINT(LEN(TUR.Orientation)), 
	pDest:= ADR(SendTelegram), 
	DestLen:= SIZEOF(SendTelegram), 
	WritePointer:= WritePointer);
	
F_AssembleByteStream(
	pSrc:= ADR(TUR.TU_Parameter), 
	SrcLen:= INT_TO_UDINT(LEN(TUR.TU_Parameter)), 
	pDest:= ADR(SendTelegram), 
	DestLen:= SIZEOF(SendTelegram), 
	WritePointer:= WritePointer);

F_AssembleByteStream(
	pSrc:= ADR(TUR.IO_Data), 
	SrcLen:= INT_TO_UDINT(LEN(TUR.IO_Data)), 
	pDest:= ADR(SendTelegram), 
	DestLen:= SIZEOF(SendTelegram), 
	WritePointer:= WritePointer);

F_AssembleByteStream(
	pSrc:= ADR(TUR.LowerLimit), 
	SrcLen:= INT_TO_UDINT(LEN(TUR.LowerLimit)), 
	pDest:= ADR(SendTelegram), 
	DestLen:= SIZEOF(SendTelegram), 
	WritePointer:= WritePointer);
	
F_AssembleByteStream(
	pSrc:= ADR(TUR.UpperLimit), 
	SrcLen:= INT_TO_UDINT(LEN(TUR.UpperLimit)), 
	pDest:= ADR(SendTelegram), 
	DestLen:= SIZEOF(SendTelegram), 
	WritePointer:= WritePointer);
	
F_AssembleByteStream(
	pSrc 			:= ADR(TUR.Sequence), 
	SrcLen 			:= INT_TO_UDINT(LEN(TUR.Sequence)), 
	pDest 			:= ADR(SendTelegram), 
	DestLen 		:= SIZEOF(SendTelegram), 
	WritePointer	:= WritePointer);
	
F_AssembleByteStream(
	pSrc 			:= ADR(TUR.SubSequence), 
	SrcLen 			:= INT_TO_UDINT(LEN(TUR.SubSequence)), 
	pDest 			:= ADR(SendTelegram), 
	DestLen 		:= SIZEOF(SendTelegram), 
	WritePointer	:= WritePointer);

F_AssembleByteStream(
	pSrc 			:= ADR(TUR.SequenceSize), 
	SrcLen 			:= INT_TO_UDINT(LEN(TUR.SequenceSize)), 
	pDest 			:= ADR(SendTelegram), 
	DestLen 		:= SIZEOF(SendTelegram), 
	WritePointer	:= WritePointer);	

F_AssembleByteStream(
	pSrc 			:= ADR(TUR.GroupID), 
	SrcLen 			:= INT_TO_UDINT(LEN(TUR.GroupID)), 
	pDest 			:= ADR(SendTelegram), 
	DestLen 		:= SIZEOF(SendTelegram), 
	WritePointer	:= WritePointer);	

F_AssembleByteStream(
	pSrc 			:= ADR(TUR.GroupSize), 
	SrcLen 			:= INT_TO_UDINT(LEN(TUR.GroupSize)), 
	pDest 			:= ADR(SendTelegram), 
	DestLen 		:= SIZEOF(SendTelegram), 
	WritePointer	:= WritePointer);	

F_AssembleByteStream(
	pSrc 			:= ADR(TUR.DestinationSlot), 
	SrcLen 			:= INT_TO_UDINT(LEN(TUR.DestinationSlot)), 
	pDest 			:= ADR(SendTelegram), 
	DestLen 		:= SIZEOF(SendTelegram), 
	WritePointer	:= WritePointer);	
	
F_AssembleByteStream(
	pSrc:= ADR(TUR.ReturnCode), 
	SrcLen:= INT_TO_UDINT(LEN(TUR.ReturnCode)), 
	pDest:= ADR(SendTelegram), 
	DestLen:= SIZEOF(SendTelegram), 
	WritePointer:= WritePointer);

F_AssembleByteStream(
	pSrc:= ADR(TUR.NumberOfDestinations), 
	SrcLen:= INT_TO_UDINT(LEN(TUR.NumberOfDestinations)), 
	pDest:= ADR(SendTelegram), 
	DestLen:= SIZEOF(SendTelegram), 
	WritePointer:= WritePointer);

// Get Destinations 
FOR DestinationIdx := 1 TO TUR_ITC.NumberOfDestinations DO
	F_AssembleByteStream(
		pSrc:= ADR(TUR.Destination[DestinationIdx]), 
		SrcLen:= INT_TO_UDINT(LEN(TUR.Destination[DestinationIdx])), 
		pDest:= ADR(SendTelegram), 
		DestLen:= SIZEOF(SendTelegram), 
		WritePointer:= WritePointer);
END_FOR

// Add to buffer of Base Driver
M_ProcessTUR := fbBaseDriver.M_SendAppData(
					mpSendData := ADR(SendTelegram),
					mSendDataLen := WritePointer);

// Forward to mirror channel
M_MirrorData(Data := ADR(SendTelegram), DataLen := WritePointer);
END_METHOD

METHOD PROTECTED M_ProcessVIR : BOOL
(**************************************************************************************
 * 	Application		:	BoxControl Framework
 *	Revision		:	$Revision: 404529 $
 *	Revision date	:	$Date: 2018-04-23 08:21:38 +0200 (Mo., 23 Apr 2018) $
 *	Last changed by	:	$Author: b7bolm $
 *	URL				:	$URL: http://almscdc.swisslog.com/repo/SWPD/Development/BoxControlFramework/20_Release/trunk/01_Software/BCF/BCF/JumpStart/20_Product/10_App/11_Com/10_Lib/10_Conv/12_MFCS/11_SIS/FB_SIS_MsgManager_6_1.TcPOU $
 *
 *	Purpose			:	Send POR
 *
 * ------------------------------------------------------------------------------------
 *	Copyright Swisslog [IP AG], Switzerland. All rights reserved.
 * 
 * ------------------------------------------------------------------------------------
 *	
 * 	Revision History: 
 *
 * 	VERSION			DATE			INITIALS			DESCRIPTION
 *	0.1				01.01.2001		swl					Example
 *
 **************************************************************************************)
VAR_INPUT
 	meChannelSrc		: E_MFCS_Channel; // Source communicaton channel
	mpVIR				: POINTER TO ST_ITC_VIR; // Pointer to POR
END_VAR

VAR
	Idx					: INT;
END_VAR
(**************************************************************************************************************
 	Check if a telegram needs to be send
***************************************************************************************************************)
// If settings allow sending a VIR 	
IF  Settings.Telegrams.SendVIR THEN
	// If the source of the request is this channel or is undefined
	IF meChannelSrc = Settings.MFCS_Channel OR
		meChannelSrc = E_MFCS_Channel.BEGIN_CHANNEL THEN
		;//Proceed
	ELSE // Source is a different MFCS Connection
		// Dont send a telegram		
		RETURN;
	END_IF	
ELSE
	// Dont send a telegram		
	RETURN;
END_IF

(**************************************************************************************************************
 	ITC - Map generic data to type
***************************************************************************************************************)
MEMCPY(destAddr := ADR(VIR_ITC), srcAddr := mpVIR, n := SIZEOF(VIR_ITC));

(**************************************************************************************************************
 	Formatting data
***************************************************************************************************************)

// Get SIS-Number 
VIR.Position := F_StuffString(
					InputString 	:= VIR_ITC.Position, 
					StringLength	:= SIS_6_1.POSITION_STRINGLENGTH, 
					StuffCharacter 	:= '0',
					LeftAligned		:= FALSE);

// Get Number of key value pairs 
VIR.NumberOfKeyValuePairs := F_StuffString(
							InputString 	:= INT_TO_STRING(VIR_ITC.NumOfKeyValuePairs), 
							StringLength	:= SIS_6_1.VIR_NUM_OF_KEYVALUEPAIRS_STRINGLENGTH, 
							StuffCharacter 	:= '0',
							LeftAligned		:= FALSE);

// Get KeyValuePairs 
FOR Idx := 1 TO VIR_ITC.NumOfKeyValuePairs BY 1 DO
	VIR.KeyValuePairs[Idx].Key	:= F_StuffString(
									InputString		:= VIR_ITC.KeyValuePair[Idx].Key,
									StringLength	:= SIS_6_1.VIR_KEY_STRINGLENGTH,
									StuffCharacter	:= ' ',
									LeftAligned		:= FALSE);
	
	VIR.KeyValuePairs[Idx].Value	:= F_StuffString(
										InputString		:= VIR_ITC.KeyValuePair[Idx].Value,
										StringLength	:= SIS_6_1.VIR_VALUE_STRINGLENGTH,
										StuffCharacter	:= ' ',
										LeftAligned		:= FALSE);
END_FOR

(**************************************************************************************************************
 	Build string and add to Base Driver
***************************************************************************************************************)
MEMSET(destAddr := ADR(SendTelegram), 0, SIZEOF(SendTelegram));
WritePointer := 0;

F_AssembleByteStream(
	pSrc:= ADR('VIR'),
	SrcLen:= 3,
	pDest:= ADR(SendTelegram),
	DestLen:= SIZEOF(SendTelegram),
	WritePointer:= WritePointer);
	
F_AssembleByteStream(
	pSrc:= ADR(VIR.Position), 
	SrcLen:= INT_TO_UDINT(LEN(VIR.Position)), 
	pDest:= ADR(SendTelegram), 
	DestLen:= SIZEOF(SendTelegram), 
	WritePointer:= WritePointer);
	
F_AssembleByteStream(
	pSrc:= ADR(VIR.NumberOfKeyValuePairs), 
	SrcLen:= INT_TO_UDINT(LEN(VIR.NumberOfKeyValuePairs)), 
	pDest:= ADR(SendTelegram), 
	DestLen:= SIZEOF(SendTelegram), 
	WritePointer:= WritePointer);	
	

// Add key value pairs
FOR Idx := 1 TO VIR_ITC.NumOfKeyValuePairs BY 1 DO
	F_AssembleByteStream(
		pSrc:= ADR(VIR.KeyValuePairs[Idx].Key), 
		SrcLen:= INT_TO_UDINT(LEN(VIR.KeyValuePairs[Idx].Key)), 
		pDest:= ADR(SendTelegram), 
		DestLen:= SIZEOF(SendTelegram), 
		WritePointer:= WritePointer);	
	
	F_AssembleByteStream(
		pSrc:= ADR(VIR.KeyValuePairs[Idx].Value), 
		SrcLen:= INT_TO_UDINT(LEN(VIR.KeyValuePairs[Idx].Value)), 
		pDest:= ADR(SendTelegram), 
		DestLen:= SIZEOF(SendTelegram), 
		WritePointer:= WritePointer);	
END_FOR

// Add to buffer of Base Driver
M_ProcessVIR := fbBaseDriver.M_SendAppData(
					mpSendData := ADR(SendTelegram),
					mSendDataLen := WritePointer);

// Forward to mirror channel
M_MirrorData(Data := ADR(SendTelegram), DataLen := WritePointer);
END_METHOD

METHOD M_PutMSG 
(**************************************************************************************
 * 	Application		:	BoxControl Framework
 *	Revision		:	$Revision: 404529 $
 *	Revision date	:	$Date: 2018-04-23 08:21:38 +0200 (Mo., 23 Apr 2018) $
 *	Last changed by	:	$Author: b7bolm $
 *	URL				:	$URL: http://almscdc.swisslog.com/repo/SWPD/Development/BoxControlFramework/20_Release/trunk/01_Software/BCF/BCF/JumpStart/20_Product/10_App/11_Com/10_Lib/10_Conv/12_MFCS/11_SIS/FB_SIS_MsgManager_6_1.TcPOU $
 *
 *	Purpose			:	Handling received MSGs
 *
 * ------------------------------------------------------------------------------------
 *	Copyright Swisslog [IP AG], Switzerland. All rights reserved.
 * 
 * ------------------------------------------------------------------------------------
 *	
 * 	Revision History: 
 *
 * 	VERSION			DATE			INITIALS			DESCRIPTION
 *	0.1				01.01.2001		swl					Example
 *
 **************************************************************************************)
VAR_INPUT
    pData               : POINTER TO BYTE         := 0;    // Pointer to received stream
    Len                 : UDINT                   := 0;    // length of stream
END_VAR

VAR
    pString             : POINTER TO STRING       := 0;
END_VAR

(*
	This method can be overloaded to do customized
	MSG implementations.
	
	Create in project folder an FunctionBlock for
	the SIS extension.
	
	Example:
	
	1.) Create FB - FB_SIS_MsgManager6_Extended;
	2.) Extend from orginal -> Extends FB_SIS_MsgManager6_0
	3.) Copy M_PutMSG from original to your implementation
	4.) Modify M_PutMSg as you want to have it
	5.) Change in Product config the implementation to your
	    new extended SIS driver
		
*)

(*
	Example implementation:
	
	// Clear data structure 
	MEMSET(destAddr := ADR(MyMSGStructure), fillByte := 0, n := SIZEOF(MyMSGStructure));

	// Preset offset
	IdxOffset := SIS_6_0.APP_DATA_OFFSET + 1;
	
	// Get subtype '000' - '999' of MSG
	MEMCPY(destAddr := ADR(MyMSGStructure.subtype), srcAddr := pData + IdxOffset), n := LENGTH_OF_SUBTYPE);
	
	// Do the same for customized content
	.
	.
	.
	.
	.
	
	
	// If no error was happing during processing, inform the driver message was processed and send 
	// it to mirror channel for logging
	IF NoError THEN
		// Message processed
		fbBaseDriver.M_ProcessedMsg();
		
		// Forward to mirror channel
		M_MirrorData(Data := pData, DataLen := Len);
	END_IF
*)



//_______________________________________________________________________________________
// if not overloaded, dump telegram and create a debug message
fbBaseDriver.M_ProcessedMsg();

// example: 'AM TCP/IP Driver,  customized MSG telegram implementation missing,  telegram = MSG987_THE_ANSWER_IS_42_ALWAYS'
DebugMsg:= '';
DebugMsg:= CONCAT(DebugMsg, Settings.BaseDriver.TCP_Driver.ChannelName);
DebugMsg:= CONCAT(DebugMsg, ',  customized MSG telegram implementation missing');
//-- telegram -----------------------------------
pString:= pData;
IF pString <> 0 THEN
    DebugMsg:= CONCAT(DebugMsg, DebugTextBlocks.TELEGRAM);
    DebugMsg:= CONCAT(DebugMsg, pString^);
END_IF

//-- send it ------------------------------------
fbDebugMsg.M_SendErrorMsg(DebugMsg);
END_METHOD

METHOD M_SendAppData : BOOL
(**************************************************************************************
 * 	Application		:	BoxControl Framework
 *	Revision		:	$Revision: 404529 $
 *	Revision date	:	$Date: 2018-04-23 08:21:38 +0200 (Mo., 23 Apr 2018) $
 *	Last changed by	:	$Author: b7bolm $
 *	URL				:	$URL: http://almscdc.swisslog.com/repo/SWPD/Development/BoxControlFramework/20_Release/trunk/01_Software/BCF/BCF/JumpStart/20_Product/10_App/11_Com/10_Lib/10_Conv/12_MFCS/11_SIS/FB_SIS_MsgManager_6_1.TcPOU $
 *
 *	Purpose			:	Send application data to a max length of 255
 *
 * ------------------------------------------------------------------------------------
 *	Copyright Swisslog [IP AG], Switzerland. All rights reserved.
 * 
 * ------------------------------------------------------------------------------------
 *	
 * 	Revision History: 
 *
 * 	VERSION			DATE			INITIALS			DESCRIPTION
 *	0.1				01.01.2001		swl					Example
 *
 **************************************************************************************)
 VAR_INPUT
	 pData		: PVOID;
	 DataLen	: UDINT;
 END_VAR

// Add to buffer of Base Driver
M_SendAppData := fbBaseDriver.M_SendAppData(
					mpSendData 		:= pData,
					mSendDataLen	:= DataLen);
END_METHOD

METHOD M_SendData : BOOL
(**************************************************************************************
 * 	Application		:	BoxControl Framework
 *	Revision		:	$Revision: 404529 $
 *	Revision date	:	$Date: 2018-04-23 08:21:38 +0200 (Mo., 23 Apr 2018) $
 *	Last changed by	:	$Author: b7bolm $
 *	URL				:	$URL: http://almscdc.swisslog.com/repo/SWPD/Development/BoxControlFramework/20_Release/trunk/01_Software/BCF/BCF/JumpStart/20_Product/10_App/11_Com/10_Lib/10_Conv/12_MFCS/11_SIS/FB_SIS_MsgManager_6_1.TcPOU $
 *
 *	Purpose			:	Send out
 *
 * ------------------------------------------------------------------------------------
 *	Copyright Swisslog [IP AG], Switzerland. All rights reserved.
 * 
 * ------------------------------------------------------------------------------------
 *	
 * 	Revision History: 
 *
 * 	VERSION			DATE			INITIALS			DESCRIPTION
 *	0.1				01.01.2001		swl					Example
 *
 **************************************************************************************)
VAR_INPUT
	meChannelSrc	: E_MFCS_Channel; // Source communicaton channel	
	mMsgType		: INT;
	mpData			: PVOID;
	mLen			: UDINT;
END_VAR

// Translate type to enumeration
eMsgType := mMsgType;

// Go to corresponding type
CASE eMsgType OF
	
	(**************************************************************************************
   		No message
	***************************************************************************************)
	E_ITC_MsgTypeConv.NO_MESSAGE_TYPE:
		;
		
	(**************************************************************************************
   		Robot command complete 
	***************************************************************************************)
	E_ITC_MsgTypeConv.ROBOT_ACTION_COMPLETE:
		// Process
		M_SendData := M_ProcessRAC(
							meChannelSrc := meChannelSrc,
							mpRAC := mpData);

	(**************************************************************************************
   		Robot delete report 
	***************************************************************************************)
	E_ITC_MsgTypeConv.ROBOT_ACTION_REQUEST:
		// Process
		M_SendData := M_ProcessRAQ(
							meChannelSrc := meChannelSrc,
							mpRAQ := mpData);
							
	(**************************************************************************************
   		Robot delete report 
	***************************************************************************************)
	E_ITC_MsgTypeConv.ROBOT_DELETE_REPORT:
		// Process
		M_SendData := M_ProcessRDR(
							meChannelSrc := meChannelSrc,
							mpRDR := mpData);

	(**************************************************************************************
   		Visualization information request 
	***************************************************************************************)	
	E_ITC_MsgTypeConv.VISUALIZATION_INFORMATION_REPORT:
		// Process
		M_SendData := M_ProcessVIR(
							meChannelSrc := meChannelSrc,
							mpVIR := mpData);	
		
	(**************************************************************************************
   		Element control reply
	***************************************************************************************)
	E_ITC_MsgTypeConv.ELEMENT_CONTROL_REPLY:
		// Process
		M_SendData := M_ProcessECR(
						meChannelSrc := meChannelSrc,
						mpECR		 := mpData);
		
	(**************************************************************************************
   		ELEMENT_STATUS_REPORT
	***************************************************************************************)
	E_ITC_MsgTypeConv.ELEMENT_STATUS_REPORT:
		// Process
		M_SendData := M_ProcessESR(
						meChannelSrc := meChannelSrc,
						mpESR		 := mpData);
		
	(**************************************************************************************
   		FUNCTION_CONTROL_REPLY
	***************************************************************************************)
	E_ITC_MsgTypeConv.FUNCTION_CONTROL_REPLY:
		// Process
		M_SendData := M_ProcessFCR(
						meChannelSrc := meChannelSrc,
						mpFCR		 := mpData);
		
	(**************************************************************************************
   		FUNCTION_STATUS_REPORT
	***************************************************************************************)
	E_ITC_MsgTypeConv.FUNCTION_STATUS_REPORT:
		// Process
		M_SendData := M_ProcessFSR(
						meChannelSrc := meChannelSrc,
						mpFSR		 := mpData);
		
	(**************************************************************************************
   		GROUP_CONTROL_REPLY
	***************************************************************************************)
	E_ITC_MsgTypeConv.GROUP_CONTROL_REPLY:
		// Process
		M_SendData := M_ProcessGCR(
						meChannelSrc := meChannelSrc,
						mpGCR		 := mpData);
		
	(**************************************************************************************
   		GROUP_STATUS_REPORT
	***************************************************************************************)
	E_ITC_MsgTypeConv.GROUP_STATUS_REPORT:
		// Process
		M_SendData := M_ProcessGSR(
						meChannelSrc := meChannelSrc,
						mpGSR		 := mpData);
		
	(**************************************************************************************
   		GLOBAL_VARIABLE_REPORT
	***************************************************************************************)
	E_ITC_MsgTypeConv.GLOBAL_VARIABLE_REPORT:
		// Process
		M_SendData := M_ProcessGVR(
						meChannelSrc := meChannelSrc,
						mpGVR		 := mpData);
		
	(**************************************************************************************
   		IDENTIFICATION_REPORT
	***************************************************************************************)
	E_ITC_MsgTypeConv.IDENTIFICATION_REPORT:
		// Process
		M_SendData := M_ProcessIPR(
						meChannelSrc := meChannelSrc,
						mpIPR		 := mpData);
		
	(**************************************************************************************
   		I_O_STATUS_REPORT
	***************************************************************************************)
	E_ITC_MsgTypeConv.I_O_STATUS_REPORT:
		// Process
		M_SendData := M_ProcessISR(
						meChannelSrc := meChannelSrc,
						mpISR		 := mpData);
		
	(**************************************************************************************
   		MANUAL_CONTROL_REPORT
	***************************************************************************************)
	E_ITC_MsgTypeConv.MANUAL_CONTROL_REPORT:
		// Process
		M_SendData := M_ProcessMCR(
						meChannelSrc := meChannelSrc,
						mpMCR		 := mpData);
		
	(**************************************************************************************
   		POSITION_OCCUPIED_REPORT
	***************************************************************************************)
	E_ITC_MsgTypeConv.POSITION_OCCUPIED_REPORT:
		// Process
		M_SendData := M_ProcessPOR(
						meChannelSrc := meChannelSrc,
						mpPOR		 := mpData);
	
	(**************************************************************************************
   		SUBSYSTEM_CONTROL_REPLY
	***************************************************************************************)
	E_ITC_MsgTypeConv.SUBSYSTEM_CONTROL_REPLY:
		// Process
		M_SendData := M_ProcessSCR(
						meChannelSrc := meChannelSrc,
						mpSCR		 := mpData);
		
	(**************************************************************************************
   		SEND_DIGITAL_INPUT
	***************************************************************************************)
	E_ITC_MsgTypeConv.SEND_DIGITAL_INPUT:
		// Process
		M_SendData := M_ProcessSDI(
						meChannelSrc := meChannelSrc,
						mpSDI		 := mpData);
		
	(**************************************************************************************
   		SCANNER_INFORMATION_REPORT
	***************************************************************************************)
	E_ITC_MsgTypeConv.SCANNER_INFORMATION_REPORT:
		// Process
		M_SendData := M_ProcessSIR(
						meChannelSrc := meChannelSrc,
						mpSIR		 := mpData);
		
	(**************************************************************************************
   		SCANNER_NO_READ_REPORT
	***************************************************************************************)
	E_ITC_MsgTypeConv.SCANNER_NO_READ_REPORT:
		// Process
		M_SendData := M_ProcessSNR(
						meChannelSrc := meChannelSrc,
						mpSNR		 := mpData);
		
	(**************************************************************************************
   		SUBSYSTEM_STATUS_REPORT
	***************************************************************************************)
	E_ITC_MsgTypeConv.SUBSYSTEM_STATUS_REPORT:
		// Process
		M_SendData := M_ProcessSSR(
						meChannelSrc := meChannelSrc,
						mpSSR		 := mpData);
		
	(**************************************************************************************
   		TASK_DELETE_REPORT
	***************************************************************************************)
	E_ITC_MsgTypeConv.TASK_DELETE_REPORT:
		// Process
		M_SendData := M_ProcessTDR(
						meChannelSrc := meChannelSrc,
						mpTDR		 := mpData);
		
	(**************************************************************************************
   		TRANSPORT_TASK_COMPLETE
	***************************************************************************************)
	E_ITC_MsgTypeConv.TRANSPORT_TASK_COMPLETE:
		// Process
		M_SendData := M_ProcessTTC(
						meChannelSrc := meChannelSrc,
						mpTTC		 := mpData);
		
	(**************************************************************************************
   		TRANSPORT_TASK_REQUEST
	***************************************************************************************)
	E_ITC_MsgTypeConv.TRANSPORT_TASK_REQUEST:
		// Process
		M_SendData := M_ProcessTTQ(
						meChannelSrc := meChannelSrc,
						mpTTQ		 := mpData);
		
	(**************************************************************************************
   		TRANSPORT_UNIT_REPORT
	***************************************************************************************)
	E_ITC_MsgTypeConv.TRANSPORT_UNIT_REPORT:
		// Process
		M_SendData := M_ProcessTUR(
						meChannelSrc := meChannelSrc,
						mpTUR		 := mpData);
		
	(**************************************************************************************
   		DATA_ACQUISITION_REPORT
	***************************************************************************************)
	E_ITC_MsgTypeConv.DATA_ACQUISITION_REPORT:
		// Process
		M_SendData := M_ProcessDAR(
						meChannelSrc := meChannelSrc,
						mpDAR		 := mpData);
		
	(**************************************************************************************
   		GATHERED_DATA_REPORT
	***************************************************************************************)
	E_ITC_MsgTypeConv.GATHERED_DATA_REPORT:
			// Process
		M_SendData := M_ProcessGDR(
						meChannelSrc := meChannelSrc,
						mpGDR		 := mpData);
		
		
	(**************************************************************************************
   		Emulation ADD TU REPORT
	***************************************************************************************)
	E_ITC_MsgTypeConv.E_ADD_TU_REPORT:
		// Process
		M_SendData := M_ProcessATR(
						meChannelSrc := meChannelSrc,
						mpATR		 := mpData);
		
	(**************************************************************************************
   		E_REMOVE_TU_REPORT
	***************************************************************************************)
	E_ITC_MsgTypeConv.E_REMOVE_TU_REPORT:
		// Process
		M_SendData := M_ProcessRTR(
						meChannelSrc := meChannelSrc,
						mpRTR		 := mpData);
		
	(**************************************************************************************
   		E_ERROR_REPORT
	***************************************************************************************)
	E_ITC_MsgTypeConv.E_ERROR_REPORT:
		// Process
		M_SendData := M_ProcessERR(
						meChannelSrc := meChannelSrc,
						mpERR		 := mpData);
						
	(**************************************************************************************
   		E_ERROR_REPORT
	***************************************************************************************)
	E_ITC_MsgTypeConv.DATA_MESSAGE:
		// Process
		M_SendData := M_SendAppData(
						pData := mpData,
						DataLen := mLen);
										
ELSE
	// Unknown type
	DebugMsg := 'Unknown message type received';
	fbDebugMsg.M_SendErrorMsg(mMessage := DebugMsg);		
END_CASE
END_METHOD

END_FUNCTION_BLOCK

(* stored: Version 1.1.0.1, ProductVersion 3.1.4024.4
   POU FB_SIS_MsgManager_6_1: Id {13243d86-7775-4b5e-be49-0d0a7c5c1419}, SpecialFunc None
   Action A_PutDAQ: Id {41605e2f-b88c-4295-8651-d46fa79fbca5}
   Action A_PutDIQ: Id {bfedb1f2-c842-4f86-b170-dca610276eb1}
   Action A_PutECQ: Id {918c7709-0a4c-44bb-96e6-dd94b0fcfece}
   Action A_PutESQ: Id {03c15598-9a40-491b-8227-33c89b4808b8}
   Action A_PutFCQ: Id {6f113aee-9fb1-43b9-b80e-46e9ad45e1f2}
   Action A_PutFSQ: Id {929a2155-37a7-4c5a-83b4-9166bb8c48ee}
   Action A_PutGCQ: Id {930d2b6d-dd9f-4034-be7c-7653fef374da}
   Action A_PutGDQ: Id {afc83614-788f-4076-be97-4e4be201516e}
   Action A_PutGSQ: Id {fc7f4730-3fcc-4185-ad77-fae63449cc66}
   Action A_PutGVQ: Id {9c435695-b99d-426e-aada-936c93960342}
   Action A_PutIRQ: Id {1c751583-5a32-4adb-9b62-be07fcefe86a}
   Action A_PutMCQ: Id {f1c6eb69-51f1-48b3-b223-d0b576515f83}
   Action A_PutRAA: Id {e6a9bf7d-4621-448d-8a46-4a175aa9fa7f}
   Action A_PutRDQ: Id {0413eb5f-0f74-4b9a-bb0b-88f3ea671b41}
   Action A_PutSCQ: Id {194cadb1-eedc-4bf6-8d8d-e55db626800a}
   Action A_PutSDO: Id {f2a13a5c-4030-4ebb-8d97-e4e9ac222d7c}
   Action A_PutSIQ: Id {2568d527-9cb0-411c-90a2-a8d0cca209dd}
   Action A_PutSSQ: Id {86677b49-9706-4183-b307-9866ca8d5595}
   Action A_PutTDQ: Id {0746988b-56f5-45fc-ba7e-fd089e1dcfda}
   Action A_PutTTA: Id {1e39672d-0814-45b2-8a2e-10c344e7b886}
   Action A_PutTUQ: Id {a0390451-940b-4230-b127-34dc30267ad8}
   Action A_PutVIQ: Id {44f0a33f-b862-43c2-9f30-0b9347e90e1c}
   Method M_BufferLevelAlarm: Id {f72202f1-fe75-4831-ac27-20ee41722c94}
   Method M_BufferLevelWarning: Id {b4ada018-004e-428b-99e9-09f301c864cd}
   Method M_CallCommunicationService: Id {f850e7bf-28b0-4355-8307-4fb9d0fe2287}
   Method M_GetReceivedData: Id {51df2264-190a-472a-8d52-3b902997a9f0}
   Method M_Init: Id {176eaacb-234a-4b3c-bdf4-46a022547e72}
   Method M_IsConnected: Id {c7577e71-a4b4-4f7d-9540-ea9da72d766d}
   Method M_MirrorData: Id {01f3e754-d4f5-406c-9401-365070a15446}
   Method M_ProcessATR: Id {4ea5f4b2-d96e-489e-a936-5ddf7d308b49}
   Method M_ProcessDAR: Id {70385093-ca52-41e4-95e9-b76bec31fb68}
   Method M_ProcessECR: Id {9c621289-e3d6-4215-8d35-66e7f4ac6c2e}
   Method M_ProcessERR: Id {1a863a9f-ee1f-4c90-85a4-03ae699abb22}
   Method M_ProcessESR: Id {9b303344-513e-4711-a44c-b38d4b43c12a}
   Method M_ProcessFCR: Id {92b37786-9860-49b1-8004-4a629704b002}
   Method M_ProcessFSR: Id {36eba689-3967-4653-813a-bf8be501b580}
   Method M_ProcessGCR: Id {0f4c9bb8-1f3e-4149-98f2-c2ec49172d7b}
   Method M_ProcessGDR: Id {23ea8b94-c5d1-4db6-948e-ea5daa9351f2}
   Method M_ProcessGSR: Id {7ece919e-443e-4c81-81ad-690220d1fb31}
   Method M_ProcessGVR: Id {b04e93ff-0c7f-408e-933f-58c6b3708e2f}
   Method M_ProcessIPR: Id {74778381-1cae-45d2-acdc-05c69e3a2860}
   Method M_ProcessISR: Id {219d441c-35dd-4595-9aa7-8702a7480f9f}
   Method M_ProcessMCR: Id {74d5f4ea-0875-484c-9c8b-8122871d91f2}
   Method M_ProcessPOR: Id {acba4193-ffdd-4e04-bb1e-51ff25dec88c}
   Method M_ProcessRAC: Id {635ff728-583e-4131-a556-110ba0339a16}
   Method M_ProcessRAQ: Id {55716850-3f57-4596-9aa2-d5bdfff718ac}
   Method M_ProcessRDR: Id {28a29b5e-7092-4ef0-b883-7e3eff417f14}
   Method M_ProcessRTR: Id {5270bc3a-964c-41c9-8c7f-aa1104c2d329}
   Method M_ProcessSCR: Id {e16160fc-b3c1-4ccf-aeab-09a2fdf8bb53}
   Method M_ProcessSDI: Id {05462b65-f04e-4cc7-8b43-376869ea7710}
   Method M_ProcessSIR: Id {734af034-00a6-4565-b3e6-13761bf8a8d2}
   Method M_ProcessSNR: Id {9dbad9e2-223a-412d-b11d-d8e97a53a42d}
   Method M_ProcessSSR: Id {769f83cf-4e3c-4450-a930-f13b288c2649}
   Method M_ProcessTDR: Id {ccebc1eb-81ff-40c4-a75a-45baba766bc4}
   Method M_ProcessTTC: Id {536aa0b3-fbe5-49a7-9fd1-cf9527381c5f}
   Method M_ProcessTTQ: Id {7006f1e6-c7de-47cf-b964-681ea2da86af}
   Method M_ProcessTUR: Id {9be0b286-ffa8-47a5-b144-f4ebba83eff5}
   Method M_ProcessVIR: Id {ca997cff-ed65-4843-8162-913b3500cc20}
   Method M_PutMSG: Id {84edc818-343b-4103-baec-5ffcaa315e62}
   Method M_SendAppData: Id {6dbd4d25-f4ca-47d3-a156-71d172c05540}
   Method M_SendData: Id {85c1dc8d-09b0-4381-9c20-3d4b6ce33410} *)
